{attribute 'linkalways'}
{attribute 'hide_all_locals'}
FUNCTION_BLOCK ValueTime EXTENDS ValueTimeRead IMPLEMENTS Value
VAR
END_VAR

METHOD SetFromType : BOOL
VAR_INPUT
	source : __SYSTEM.AnyType;
END_VAR
SetFromType := ConvertAnyType(source, thisAnyType);
END_METHOD

METHOD SetFromString : BOOL
VAR_INPUT
	value : T_MaxString;
END_VAR
thisValue := STRING_TO_TIME(value);

SetFromString := TRUE;
END_METHOD

METHOD Set : BOOL
VAR_INPUT
	source : ANY;
END_VAR
Set := ConvertAnyType(source, thisAnyType);
END_METHOD

END_FUNCTION_BLOCK

(* stored: Version 1.1.0.1
   POU ValueTime: Id {1f55a405-48d4-4799-90bc-d667bb4af4a7}, SpecialFunc None
   Method SetFromType: Id {718a89d4-10a9-4803-8488-33f4af29bbd6}
   Method SetFromString: Id {3f3e88b4-3323-445b-8049-1cd4a349f528}
   Method Set: Id {90274564-48dd-476f-84f3-e8565819c03d} *)
